PROGRAM MAIN
VAR
	// print out 'Hello world'
	fbStringBuilder : FB_StringBuilder;
	sResult : STRING;
	bTest : BOOL;
END_VAR

IF bTest THEN
	sResult := fbStringBuilder.Clear()^
								.Append('H')^
								.Append('e')^
								.Append('l')^
								.Append('l')^
								.Append('o')^
								.Append(' ')^
								.Append('W')^
								.Append('o')^
								.Append('r')^
								.Append('l')^
								.Append('d')^
								.ToString();
	bTest := FALSE;
END_IF

END_PROGRAM

(* stored: Version 1.1.0.1, ProductVersion 3.1.4024.12
   POU MAIN: Id {858ed81e-6f93-475b-bad7-626407de5004}, SpecialFunc None *)
